(* LS Electric XG5000 project: imports *)
(* PLC LSPLC *)

FUNCTION_BLOCK 오초깜빡이
VAR_INPUT
    FL : BOOL;
    NFL : BOOL;
    OFF : BOOL;
END_VAR
VAR_OUTPUT
    출력1 : BOOL;
    출력2 : BOOL;
END_VAR
VAR
    FL자가유지 : BOOL;
    NFL자가유지 : BOOL;
    타이머1 : TP;
    타이머2 : TP;
END_VAR

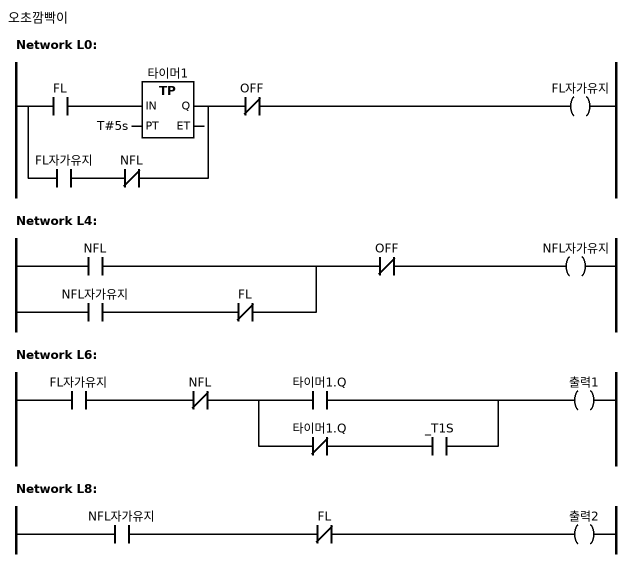
(* Rung L0 *)
타이머1(IN := FL, PT := T#5s);
FL자가유지 := (타이머1.Q OR (FL자가유지 AND NOT NFL)) AND NOT OFF;
(* Rung L4 *)
NFL자가유지 := (NFL OR (NFL자가유지 AND NOT FL)) AND NOT OFF;
(* Rung L6 *)
출력1 := FL자가유지 AND NOT NFL AND (타이머1.Q OR (NOT 타이머1.Q AND _T1S));
(* Rung L8 *)
출력2 := NFL자가유지 AND NOT FL;
END_FUNCTION_BLOCK

PROGRAM NewProgram (* task: 스캔 프로그램 *)
VAR
    FL : BOOL;
    NFL : BOOL;
    OFF : BOOL;
    깜빡이 : 오초깜빡이;
END_VAR

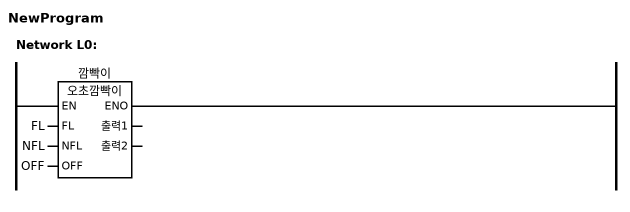
(* Rung L0 *)
깜빡이(FL := FL, NFL := NFL, OFF := OFF);
END_PROGRAM